(* LS Electric XG5000 project: XGB_TemperatureMeasuring *)
(* XGB temperature measuring example program *)
(* PLC LSPLC *)
(* module base 0 slot 0: Input/Output Module:XEM-DN/DP32HP (DC 24V Input, Transistor Output, 32 Contacts) *)
(* module base 0 slot 1: Internal Positioning:XBF-PO06E (Open Collector Type, 6 Axis) *)
(* module base 0 slot 2: Temp. Measuring Module:XBF-TC04S (Temperature Input Type(4 Channels)) *)
VAR_GLOBAL
    _02_CH0_ACT AT %UX0.2.16 : BOOL; (* Temp. Measuring Module : CH0 Activation Status *)
    _02_CH0_BOUT AT %UX0.2.20 : BOOL; (* Temp. Measuring Module : CH0 Disconnection Flag *)
    _02_CH0_SETERR AT %UX0.2.24 : BOOL; (* Temp. Measuring Module : CH0 Error Code *)
    _02_CH0_TEMP AT %UW0.2.4 : WORD; (* Temp. Measuring Module : CH0 Temp. Data *)
    _02_CH_ADJERR_ARY AT %UX0.2.0 : ARRAY[0..3] OF BOOL; (* Temp. Measuring Module : Each CH Offset/Gain Error Flag *)
    _02_RDY AT %UX0.2.15 : BOOL; (* Temp. Measuring Module : Ready Flag *)
    _02_WDT_ERR AT %UX0.2.14 : BOOL; (* Temp. Measuring Module : H/W Error Flag *)
END_VAR

PROGRAM TemperatureMeasuring (* task: Scan Program *)
VAR
    CH0_Disconnected : BOOL; (* Channel 0 disconnected error status *)
    CH0_Temperature : INT; (* Channel 0 temperature value *)
    Temp_CH0_Ready : BOOL; (* Channel 0 is ready *)
END_VAR
VAR_EXTERNAL
    _02_CH0_ACT : BOOL; (* AT %UX0.2.16 *) (* Temp. Measuring Module : CH0 Activation Status *)
    _02_CH0_BOUT : BOOL; (* AT %UX0.2.20 *) (* Temp. Measuring Module : CH0 Disconnection Flag *)
    _02_CH0_SETERR : BOOL; (* AT %UX0.2.24 *) (* Temp. Measuring Module : CH0 Error Code *)
    _02_CH0_TEMP : WORD; (* AT %UW0.2.4 *) (* Temp. Measuring Module : CH0 Temp. Data *)
    _02_CH_ADJERR_ARY : ARRAY[0..3] OF BOOL; (* AT %UX0.2.0 *) (* Temp. Measuring Module : Each CH Offset/Gain Error Flag *)
    _02_RDY : BOOL; (* AT %UX0.2.15 *) (* Temp. Measuring Module : Ready Flag *)
    _02_WDT_ERR : BOOL; (* AT %UX0.2.14 *) (* Temp. Measuring Module : H/W Error Flag *)
END_VAR

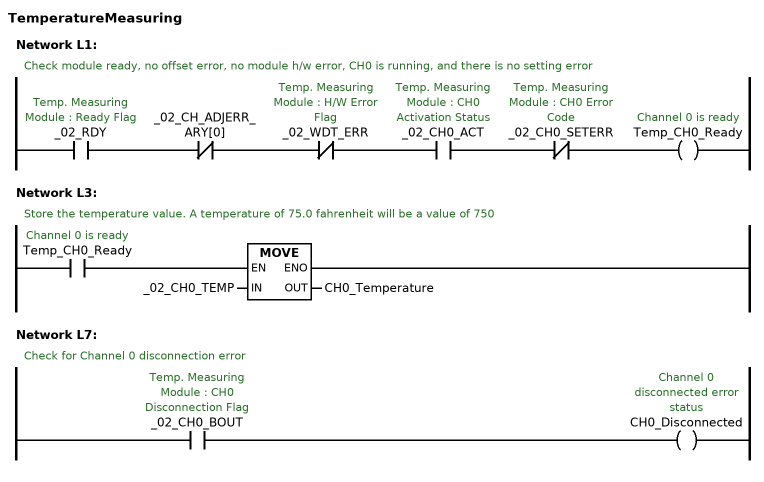
(* Check module ready, no offset error, no module h/w error, CH0 is running, and there is no setting error *)
(* Rung L1 *)
Temp_CH0_Ready := _02_RDY AND NOT _02_CH_ADJERR_ARY[0] AND NOT _02_WDT_ERR AND _02_CH0_ACT AND NOT _02_CH0_SETERR;
(* Store the temperature value. A temperature of 75.0 fahrenheit will be a value of 750 *)
(* Rung L3 *)
IF Temp_CH0_Ready THEN CH0_Temperature := _02_CH0_TEMP; END_IF;
(* Check for Channel 0 disconnection error *)
(* Rung L7 *)
CH0_Disconnected := _02_CH0_BOUT;
END_PROGRAM